FUNCTION_BLOCK FB_UN_base
VAR
	TagName : STRING;
	Description : STRING;
	TagID : INT;
END_VAR

END_FUNCTION_BLOCK

(* stored: Version 1.1.0.1, ProductVersion 3.1.4024.12
   POU FB_UN_base: Id {0ff46b31-ca57-435d-9419-c972abdcf761}, SpecialFunc None *)
